(* PLC project SafeLOGIC, BrAutomation SafeDESIGNER  5.24.1.0 *)
(* stored: companyURL http://www.br-automation.com, creationDateTime Wed Dec 10 18:10:20 2025 *)

PROGRAM Main
  VAR  (* added by the conversion: wires and edge detectors of the diagram *)
    _SEL_S37_OUT : SAFEDINT;
  END_VAR

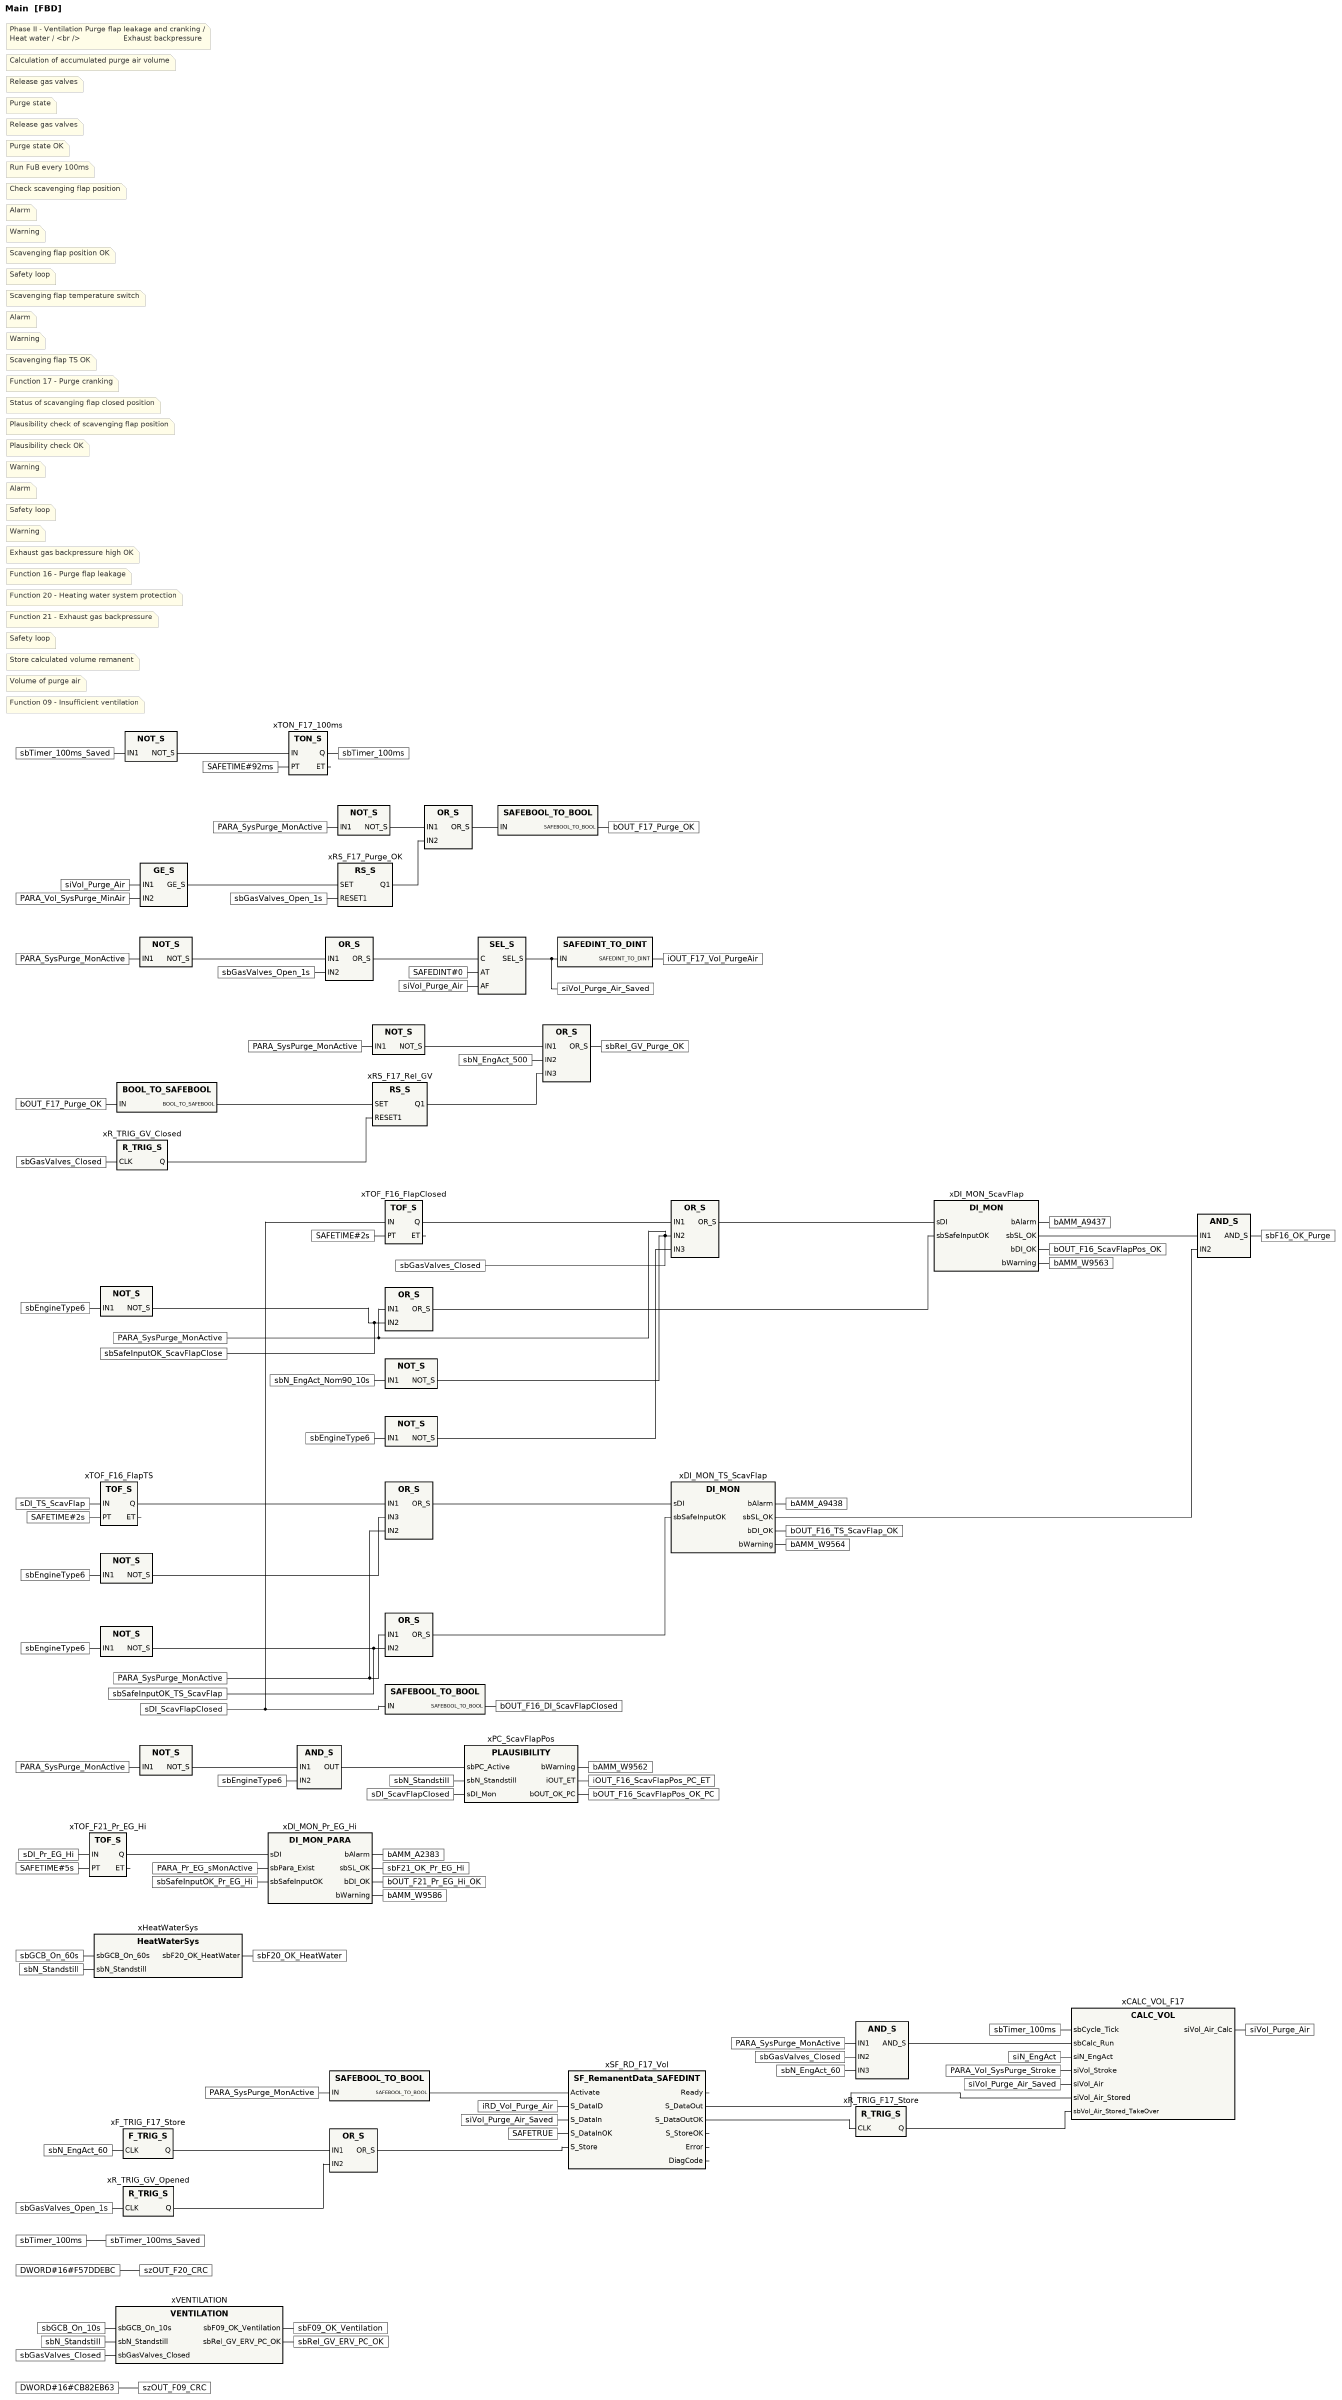
(* FBD diagram, written out as Structured Text *)
(* Phase II - Ventilation Purge flap leakage and cranking / Heat water / <br />                   Exhaust backpressure *)
(* Function 09 - Insufficient ventilation *)
xVENTILATION(sbGCB_On_10s := sbGCB_On_10s, sbN_Standstill := sbN_Standstill, sbGasValves_Closed := sbGasValves_Closed);
sbF09_OK_Ventilation := xVENTILATION.sbF09_OK_Ventilation;
sbRel_GV_ERV_PC_OK := xVENTILATION.sbRel_GV_ERV_PC_OK;
szOUT_F09_CRC := DWORD#16#CB82EB63;
(* Function 16 - Purge flap leakage *)
(* Check scavenging flap position *)
(* Status of scavanging flap closed position *)
bOUT_F16_DI_ScavFlapClosed := SAFEBOOL_TO_BOOL(sDI_ScavFlapClosed);
(* Alarm *)
xTOF_F16_FlapClosed(IN := sDI_ScavFlapClosed, PT := SAFETIME#2s);
xDI_MON_ScavFlap(sDI := OR_S(xTOF_F16_FlapClosed.Q, NOT_S(sbN_EngAct_Nom90_10s), NOT_S(sbEngineType6), sbGasValves_Closed, PARA_SysPurge_MonActive), sbSafeInputOK := OR_S(PARA_SysPurge_MonActive, NOT_S(sbEngineType6), sbSafeInputOK_ScavFlapClose));
bAMM_A9437 := xDI_MON_ScavFlap.bAlarm;
(* Scavenging flap position OK *)
(* Warning *)
bAMM_W9563 := xDI_MON_ScavFlap.bWarning;
bOUT_F16_ScavFlapPos_OK := xDI_MON_ScavFlap.bDI_OK;
(* Safety loop *)
xTOF_F16_FlapTS(IN := sDI_TS_ScavFlap, PT := SAFETIME#2s);
xDI_MON_TS_ScavFlap(sDI := OR_S(xTOF_F16_FlapTS.Q, NOT_S(sbEngineType6), PARA_SysPurge_MonActive), sbSafeInputOK := OR_S(PARA_SysPurge_MonActive, NOT_S(sbEngineType6), sbSafeInputOK_TS_ScavFlap));
sbF16_OK_Purge := AND_S(xDI_MON_ScavFlap.sbSL_OK, xDI_MON_TS_ScavFlap.sbSL_OK);
(* Scavenging flap temperature switch *)
(* Alarm *)
bAMM_A9438 := xDI_MON_TS_ScavFlap.bAlarm;
(* Scavenging flap TS OK *)
(* Warning *)
bAMM_W9564 := xDI_MON_TS_ScavFlap.bWarning;
bOUT_F16_TS_ScavFlap_OK := xDI_MON_TS_ScavFlap.bDI_OK;
(* Plausibility check of scavenging flap position *)
(* Warning *)
(* Plausibility check OK *)
xPC_ScavFlapPos(sbPC_Active := AND_S(NOT_S(PARA_SysPurge_MonActive), sbEngineType6), sbN_Standstill := sbN_Standstill, sDI_Mon := sDI_ScavFlapClosed);
bAMM_W9562 := xPC_ScavFlapPos.bWarning;
bOUT_F16_ScavFlapPos_OK_PC := xPC_ScavFlapPos.bOUT_OK_PC;
iOUT_F16_ScavFlapPos_PC_ET := xPC_ScavFlapPos.iOUT_ET;
(* Function 17 - Purge cranking *)
(* Calculation of accumulated purge air volume *)
xTON_F17_100ms(IN := NOT_S(sbTimer_100ms_Saved), PT := SAFETIME#92ms);
sbTimer_100ms := xTON_F17_100ms.Q;
sbTimer_100ms_Saved := sbTimer_100ms;
(* Run FuB every 100ms *)
xF_TRIG_F17_Store(CLK := sbN_EngAct_60);
xR_TRIG_GV_Opened(CLK := sbGasValves_Open_1s);
xSF_RD_F17_Vol(Activate := SAFEBOOL_TO_BOOL(PARA_SysPurge_MonActive), S_DataID := iRD_Vol_Purge_Air, S_DataIn := siVol_Purge_Air_Saved, S_DataInOK := SAFETRUE, S_Store := OR_S(xF_TRIG_F17_Store.Q, xR_TRIG_GV_Opened.Q));
xR_TRIG_F17_Store(CLK := xSF_RD_F17_Vol.S_DataOutOK);
xCALC_VOL_F17(sbCycle_Tick := sbTimer_100ms, sbCalc_Run := AND_S(PARA_SysPurge_MonActive, sbGasValves_Closed, sbN_EngAct_60), siN_EngAct := siN_EngAct, siVol_Stroke := PARA_Vol_SysPurge_Stroke, siVol_Air := siVol_Purge_Air_Saved, siVol_Air_Stored := xSF_RD_F17_Vol.S_DataOut, sbVol_Air_Stored_TakeOver := xR_TRIG_F17_Store.Q);
siVol_Purge_Air := xCALC_VOL_F17.siVol_Air_Calc;
(* Store calculated volume remanent *)
(* Purge state *)
(* Purge state OK *)
xRS_F17_Purge_OK(SET := GE_S(siVol_Purge_Air, PARA_Vol_SysPurge_MinAir), RESET1 := sbGasValves_Open_1s);
bOUT_F17_Purge_OK := SAFEBOOL_TO_BOOL(OR_S(NOT_S(PARA_SysPurge_MonActive), xRS_F17_Purge_OK.Q1));
(* Volume of purge air *)
_SEL_S37_OUT := SEL_S(OR_S(NOT_S(PARA_SysPurge_MonActive), sbGasValves_Open_1s), SAFEDINT#0, siVol_Purge_Air);
siVol_Purge_Air_Saved := _SEL_S37_OUT;
iOUT_F17_Vol_PurgeAir := SAFEDINT_TO_DINT(_SEL_S37_OUT);
(* Release gas valves *)
(* Release gas valves *)
xR_TRIG_GV_Closed(CLK := sbGasValves_Closed);
xRS_F17_Rel_GV(SET := BOOL_TO_SAFEBOOL(bOUT_F17_Purge_OK), RESET1 := xR_TRIG_GV_Closed.Q);
sbRel_GV_Purge_OK := OR_S(NOT_S(PARA_SysPurge_MonActive), sbN_EngAct_500, xRS_F17_Rel_GV.Q1);
(* Function 20 - Heating water system protection *)
(* Safety loop *)
xHeatWaterSys(sbGCB_On_60s := sbGCB_On_60s, sbN_Standstill := sbN_Standstill);
sbF20_OK_HeatWater := xHeatWaterSys.sbF20_OK_HeatWater;
szOUT_F20_CRC := DWORD#16#F57DDEBC;
(* Function 21 - Exhaust gas backpressure *)
(* Alarm *)
(* Safety loop *)
(* Exhaust gas backpressure high OK *)
(* Warning *)
xTOF_F21_Pr_EG_Hi(IN := sDI_Pr_EG_Hi, PT := SAFETIME#5s);
xDI_MON_Pr_EG_Hi(sDI := xTOF_F21_Pr_EG_Hi.Q, sbPara_Exist := PARA_Pr_EG_sMonActive, sbSafeInputOK := sbSafeInputOK_Pr_EG_Hi);
bOUT_F21_Pr_EG_Hi_OK := xDI_MON_Pr_EG_Hi.bDI_OK;
sbF21_OK_Pr_EG_Hi := xDI_MON_Pr_EG_Hi.sbSL_OK;
bAMM_A2383 := xDI_MON_Pr_EG_Hi.bAlarm;
bAMM_W9586 := xDI_MON_Pr_EG_Hi.bWarning;
END_PROGRAM
